FUNCTION FUN_MachineState : E_MachineState
VAR_INPUT
	Error :BOOL;
	Estop : BOOL;
	Stop :BOOL;
	Reset:BOOL;
	Start :BOOL;
	HomeBusy :BOOL;
	Homed :BOOL;
	MachineMode : E_UnitMode;
	eMachineState : E_MachineState;
END_VAR
VAR
		
END_VAR

IF Error OR EStop THEN
	eMachineState:=E_MachineState.Error;
END_IF

CASE eMachineState OF
	E_MachineState.Default :
		eMachineState:=E_MachineState.NotHomed;
	E_MachineState.NotHomed:

		IF HomeBusy THEN
			eMachineState:=E_MachineState.Homing;
		ELSIF Homed THEN
			eMachineState:=E_MachineState.Homed;
		END_IF
	
	E_MachineState.Homing:
		
		IF Homed THEN
			eMachineState:=E_MachineState.Homed;
		END_IF
	
	E_MachineState.Homed:
	
		IF MachineMode = E_UnitMode.AUTO THEN
			eMachineState:=E_MachineState.Running;
		END_IF
		IF HomeBusy THEN
			eMachineState:=E_MachineState.Homing;
		END_IF
		
	E_MachineState.Running:
	
		IF Stop THEN
			eMachineState:=E_MachineState.StandBy;
		END_IF
		
		 IF MachineMode = E_UnitMode.MANUAL THEN
			eMachineState:=E_MachineState.Homed;			
		 END_IF
		 
	E_MachineState.StandBy:
		
		IF Start THEN
			eMachineState:=E_MachineState.Running;
		END_IF
		IF MachineMode = E_UnitMode.MANUAL THEN
			eMachineState:=E_MachineState.Homed;			
		 END_IF
		 
	E_MachineState.Error:
		
		IF Reset OR NOT Error THEN
			eMachineState:=E_MachineState.StandBy;
		END_IF

END_CASE

FUN_MachineState := eMachineState ;

END_FUNCTION

(* stored: Version 1.1.0.1, ProductVersion 3.1.4024.13
   POU FUN_MachineState: Id {07e1174a-fe03-4e14-a0ba-027685cb59b3}, SpecialFunc None *)
